{attribute 'linkalways'} 
{attribute 'no_explicit_call' := 'This FB is a CLASS and must be accessed using methods or properties'}
{attribute 'enable_dynamic_creation'}
FUNCTION_BLOCK Node_ContainerType_Vector_TcVnVector4_UINT EXTENDS Node
VAR
    out : _GUID;
END_VAR

METHOD PUBLIC  Clone : I_Node
VAR
	pNode : POINTER TO Node_ContainerType_Vector_TcVnVector4_UINT;
END_VAR
pNode := __NEW(Node_ContainerType_Vector_TcVnVector4_UINT);
Clone := pNode^;
END_METHOD

METHOD FB_init : BOOL
VAR_INPUT
	bInitRetains : BOOL; // if TRUE, the retain variables are initialized (warm start / cold start)
	bInCopyCode : BOOL;  // if TRUE, the instance afterwards gets moved into the copy code (online change)
END_VAR
AddOutput('out', out);
END_METHOD

METHOD PROTECTED OnExecute
out.Value := ContainerType_Vector_TcVnVector4_UINT;
END_METHOD

END_FUNCTION_BLOCK

(* stored: Version 1.1.0.1, ProductVersion 3.1.4026.17
   POU Node_ContainerType_Vector_TcVnVector4_UINT: Id {af7b26f0-7fc5-0aaf-2dfd-68fd65fb1421}, SpecialFunc None
   Folder Constructor: Id {2abf16ae-3ff0-0de3-3937-d60cf4b94cd8}
   Method Clone: Id {edc7852b-8feb-0999-3df6-914d4e4d8fb8}
   Method FB_init: Id {7c005e4e-0e34-040e-3fea-7f516c6045fe}
   Method OnExecute: Id {16f01894-84db-0ba4-3aa6-addef087b977} *)
